TYPE ST_Alarm_Hmi :
STRUCT
	msg		: STRING(255);
	str_DT	: STRING(255);
END_STRUCT
END_TYPE

(* stored: Version 1.1.0.1, ProductVersion 3.1.4024.12
   DUT ST_Alarm_Hmi: Id {be96a815-c410-4051-b2e1-b69dfb5f4496} *)
